// TIA Portal V20 export
DATA_BLOCK "DB_SafetyStandard"   // DB20
// stored: Access Published, MemoryReserve 100
   VAR
      ToStandard : Struct
         EstopActive : Bool;
      END_STRUCT;
      PressReset : Bool;
      ToHMI : Struct
         "EstopPB -MCC001+MCC001-SF1" : Bool;
         "EstopPB -ZONA1+A1.1.1-SF1" : Bool;
         "EstopPB -ZONA1+A1.1.10-SF1" : Bool;
         "EstopPB -ZONA1+A1.2.1-SF1" : Bool;
         "EstopPB -ZONA1+B1.22.1-SF1" : Bool;
         "EstopPB -ZONA1+C1.3.1-SF1" : Bool;
         "EstopPB -ZONA1+B1.12.1-SF1" : Bool;
         "EstopPB -ZONA1+B1.15.1-SF1" : Bool;
         "EstopPB -ZONA1+B1.17.3-SF1" : Bool;
         "EstopPB -ZONA2+D1.11.1-SF1" : Bool;
         "EstopPB -ZONA2+E1.1.2-SF1" : Bool;
         "EstopPB -ZONA2+A1.10.3-SF1" : Bool;
         "EstopPB -ZONA2+A1.12.1-SF1" : Bool;
         "EstopPB -ZONA2+A1.16.8-SF1" : Bool;
         "EstopPB -ZONA2+B1.17.0-SF1" : Bool;
         "EstopPB -ZONA2+A2.4.5-SF1" : Bool;
         "EstopPB -ZONA2+G1.5.3-SF1" : Bool;
         "EstopPB -ZONA2+G1.7.1-SF1" : Bool;
         "PhaseOK -MCC001" : Bool;
      END_STRUCT;
      holdAlarmOffTimer : TON_TIME;
      holdAlarmOff : Bool;
   END_VAR
BEGIN
END_DATA_BLOCK
